// TIA Portal V17 export
// export: Created 2023-03-24T09:45:04.5136241Z, ExportSetting None, DisplayName Totally Integrated Automation Portal, DisplayVersion V17 Update 4, DisplayName TIA Portal Openness, DisplayVersion V17 Update 4, DisplayName TIA Portal Version Control Interface, DisplayVersion V17, DisplayName STEP 7 Professional, DisplayVersion V17 Update 4, DisplayName STEP 7 Safety, DisplayVersion V17, DisplayName WinCC Advanced / Unified PC, DisplayVersion V17 Update 4
FUNCTION "FC_PROVA" : Void   // FC1, LAD
TITLE = goku
{ S7_Optimized_Access := 'TRUE' }
// bigol
// stored: SetENOAutomatically false
BEGIN

REGION Network 1: DESCRIPTION
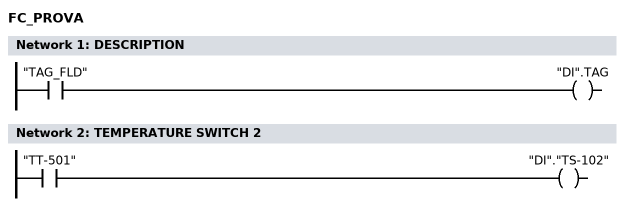
   RUNG wire#powerrail
      Contact( "TAG_FLD" )
      Coil( "DI".TAG )
   END_RUNG
   // the same network as SCL:
   "DI".TAG := "TAG_FLD";
END_REGION

REGION Network 2: TEMPERATURE SWITCH 2
   RUNG wire#powerrail
      Contact( "TT-501" )
      Coil( "DI"."TS-102" )
   END_RUNG
   // the same network as SCL:
   "DI"."TS-102" := "TT-501";
END_REGION
END_FUNCTION
